FUNCTION F_FunA : INT
VAR_INPUT
    fbMyFbA : FB_A;
END_VAR

END_FUNCTION

(* stored: Version 1.1.0.1, ProductVersion 3.1.4024.12
   POU F_FunA: Id {ac29b473-e8de-4576-a169-ecb69ef48b92}, SpecialFunc None *)
